DATA_BLOCK "ST10_Flow21_HShaftLifting_iDB"
{ S7_Optimized_Access := 'TRUE' }
VERSION : 0.1
NON_RETAIN
// ATTRIBUTES
// AUTO_NUMBER = False
// BLOCK_NUMBER = 1091
// END_ATTRIBUTES
"ST10_Flow21_HShaftLifting"

BEGIN

END_DATA_BLOCK

